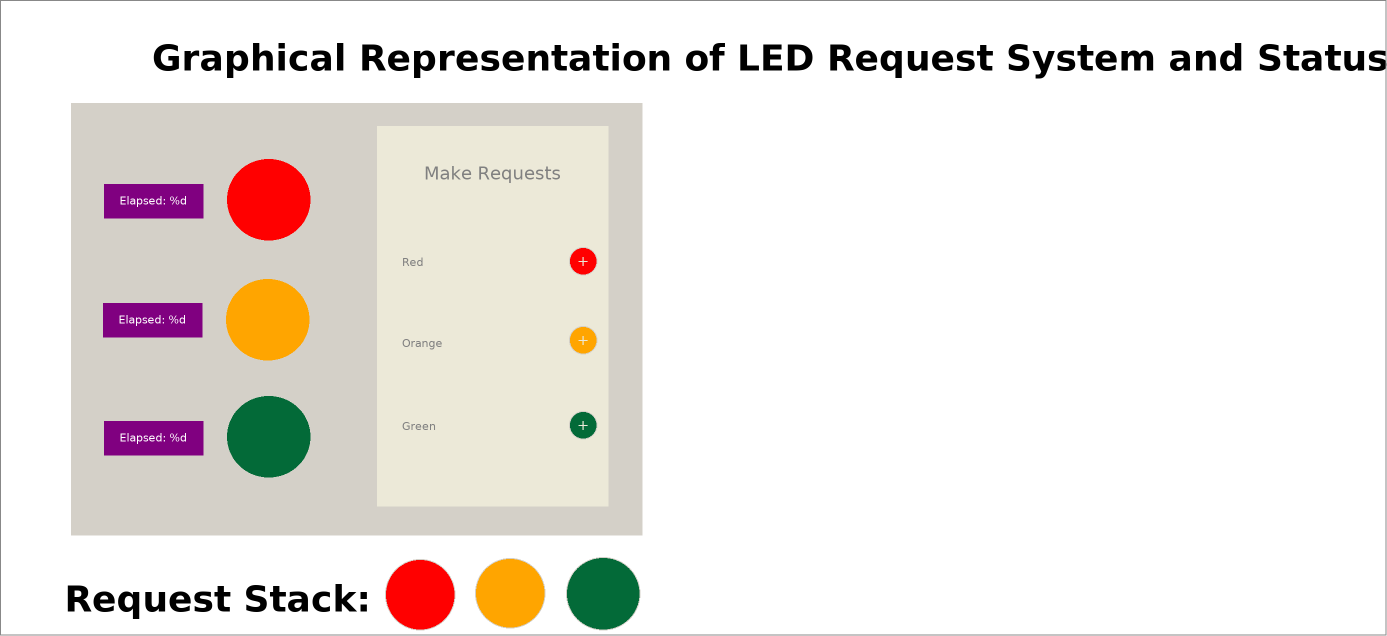
VISUALIZATION LEDUI  // 1387x636
    Label (156,23 1229x70), "Graphical Representation of LED Request System and Status"
    Rectangle (71,103 571x432)
    Ellipse (226,158 85x83)
    Ellipse (225,278 85x83)
    Ellipse (226,395 85x83)
    Rectangle (103,183 101x36), "Elapsed: %d"
    Rectangle (103,420 101x36), "Elapsed: %d"
    Rectangle (102,302 101x36), "Elapsed: %d"
    Label (39,564 358x70), "Request Stack:"
    Ellipse (385,559 70x71)
    Ellipse (475,558 70x70)
    Ellipse (566,557 74x73)
    Rectangle (376,125 233x382)
    Rectangle (381,153 223x41), "Make Requests"
    Rectangle (385,244 176x37), "Red"
    Rectangle (385,325 176x37), "Orange"
    Rectangle (385,408 176x37), "Green"
    InvisibleInput (432,248 126x30)
    InvisibleInput (447,328 111x30)
    InvisibleInput (441,412 117x30)
    Ellipse (569,247 28x28), "+"
    Ellipse (569,326 28x28), "+"
    Ellipse (569,411 28x28), "+"
END_VISUALIZATION

(* stored: Version 1.1.0.1, ProductVersion 3.1.4022.12
   Visu LEDUI: Id {50361e63-e9b3-4ac5-a954-aa49a2ec0515} *)
